PROGRAM MAIN
VAR
END_VAR

P_Task2();

END_PROGRAM

(* stored: Version 1.1.0.1, ProductVersion 3.1.4024.12
   POU MAIN: Id {d7c65d5a-4c71-432c-9b81-094e912d304b}, SpecialFunc None *)
